(* PLC project drill, Dassault Systèmes ControlBuild 2020 *)
(* stored: creationDateTime 2019-04-23T11:18:46-01:00 *)

CONFIGURATION drill
  VAR_GLOBAL
    generalPanel/powerUpPB AT 7 : BOOL := false;
    generalPanel/startCyclePB AT 8 : BOOL := false;
    generalPanel/emergencyStop AT 9 : BOOL := false;
    generalPanel/batchCycle AT 10 : BOOL := true;
    generalPanel/pieceCycle AT 11 : BOOL := false;
    generalPanel/autoSwitch AT 12 : BOOL := false;
    generalPanel/manualSwitch AT 13 : BOOL := false;
    generalPanel/acknowledgePB AT 15 : BOOL := false;
    generalPanel/powerUpPB/PB AT 7 : BOOL := false;
    generalPanel/powerUpPB/action AT 24 : BOOL := false;
    generalPanel/powerUpPB/timeCounter AT 17 : REAL := 0.0;
    generalPanel/powerUpPB/pulseDuration AT 18 : REAL := 5.0;
    generalPanel/powerUpPB/PBLogic AT 25 : BOOL := true;
    generalPanel/startCyclePB/PB AT 8 : BOOL := false;
    generalPanel/startCyclePB/action AT 26 : BOOL := false;
    generalPanel/startCyclePB/timeCounter AT 19 : REAL := 0.0;
    generalPanel/startCyclePB/pulseDuration AT 20 : REAL := 5.0;
    generalPanel/startCyclePB/PBLogic AT 27 : BOOL := true;
    generalPanel/cycleSwitch/leftVariable AT 11 : BOOL := false;
    generalPanel/cycleSwitch/rightVariable AT 10 : BOOL := true;
    generalPanel/cycleSwitch/leftPosition AT 28 : BOOL := false;
    generalPanel/cycleSwitch/rightPosition AT 29 : BOOL := false;
    generalPanel/modeSwitch/leftVariable AT 12 : BOOL := true;
    generalPanel/modeSwitch/rightVariable AT 13 : BOOL := false;
    generalPanel/modeSwitch/leftPosition AT 30 : BOOL := false;
    generalPanel/modeSwitch/rightPosition AT 31 : BOOL := false;
    generalPanel/acknowledgePB/PB AT 15 : BOOL := false;
    generalPanel/acknowledgePB/action AT 32 : BOOL := false;
    generalPanel/acknowledgePB/timeCounter AT 21 : REAL := 0.0;
    generalPanel/acknowledgePB/pulseDuration AT 22 : REAL := 5.0;
    generalPanel/acknowledgePB/PBLogic AT 33 : BOOL := true;
    generalPanel/emergencyStop/pb AT 9 : BOOL := false;
    generalPanel/emergencyStop/action AT 34 : BOOL := false;
    generalPanel/emergencyStop/PBLogic AT 35 : BOOL := false;
    workingModes/powerUpPB AT 7 : BOOL := false;
    workingModes/startCyclePB AT 8 : BOOL := false;
    workingModes/emergencyStop AT 9 : BOOL := false;
    workingModes/batchCycle AT 10 : BOOL := true;
    workingModes/pieceCycle AT 11 : BOOL := false;
    workingModes/autoSwitch AT 12 : BOOL := false;
    workingModes/manualSwitch AT 13 : BOOL := false;
    workingModes/cycleEnd AT 14 : BOOL := false;
    workingModes/acknowledgePB AT 15 : BOOL := false;
    workingModes/live AT 6 : BOOL := false;
    workingModes/autoMode AT 20 : BOOL := false;
    workingModes/manualMode AT 21 : BOOL := false;
    workingModes/emptyProd AT 17 : BOOL := false;
    workingModes/unitProd AT 18 : BOOL := false;
    workingModes/batchProd AT 19 : BOOL := false;
    workingModes/emergencyState AT 36 : BOOL := false;
    functional/piece AT 16 : BOOL := false;
    functional/emptyProd AT 17 : BOOL := false;
    functional/unitProd AT 18 : BOOL := false;
    functional/batchProd AT 19 : BOOL := false;
    functional/acknowledgePB AT 15 : BOOL := false;
    functional/autoMode AT 20 : BOOL := false;
    functional/manualMode AT 21 : BOOL := false;
    functional/faultyState AT 5 : BOOL := false;
    functional/cycleEnd AT 14 : BOOL := false;
    functional/loadingRequest AT 22 : BOOL := false;
    functional/unloadingRequest AT 23 : BOOL := false;
    functional/functionChart/rotationFault AT 529 : DINT := 0;
    functional/functionChart/downState AT 42 : BOOL := false;
    functional/functionChart/downDeceleration AT 43 : BOOL := false;
    functional/functionChart/topDeceleration AT 44 : BOOL := false;
    functional/functionChart/topState AT 45 : BOOL := false;
    functional/functionChart/motorFault AT 530 : DINT := 0;
    functional/functionChart/clampingFault AT 531 : DINT := 0;
    functional/functionChart/releasingOK AT 46 : BOOL := false;
    functional/functionChart/clampingOK AT 47 : BOOL := false;
    functional/functionChart/emptyProd AT 17 : BOOL := false;
    functional/functionChart/unitProd AT 18 : BOOL := false;
    functional/functionChart/batchProd AT 19 : BOOL := false;
    functional/functionChart/acknowledgePB AT 15 : BOOL := false;
    functional/functionChart/piece AT 16 : BOOL := false;
    functional/functionChart/rotation AT 54 : BOOL := false;
    functional/functionChart/cycleEnd AT 14 : BOOL := false;
    functional/functionChart/movementFault AT 528 : DINT := 0;
    functional/functionChart/loadingRequest AT 22 : BOOL := false;
    functional/functionChart/unloadingRequest AT 23 : BOOL := false;
    functional/functionChart/faultyState AT 5 : BOOL := false;
    functional/functionChart/slowAscent AT 48 : BOOL := false;
    functional/functionChart/fastAscent AT 49 : BOOL := false;
    functional/functionChart/slowDescent AT 50 : BOOL := false;
    functional/functionChart/fastDescent AT 51 : BOOL := false;
    functional/functionChart/releasing AT 52 : BOOL := false;
    functional/functionChart/clamping AT 53 : BOOL := false;
    functional/functionChart/initialCond AT 55 : BOOL := false;
    functional/functionChart/noFaultCond AT 56 : BOOL := false;
    functional/functionChart/cnt AT 532 : DINT := 0;
    functional/functionChart/_X_10 AT 57 : BOOL := true;
    functional/functionChart/_X_11 AT 58 : BOOL := false;
    functional/functionChart/_X_12 AT 59 : BOOL := false;
    functional/functionChart/_X_13 AT 60 : BOOL := false;
    functional/functionChart/_X_14 AT 61 : BOOL := false;
    functional/functionChart/_X_15 AT 62 : BOOL := false;
    functional/functionChart/_X_16 AT 63 : BOOL := false;
    functional/functionChart/_X_17 AT 64 : BOOL := false;
    functional/functionChart/fastDescentDuration AT 533 : DINT := 100;
    functional/functionChart/slowDescentDuration AT 534 : DINT := 50;
    functional/functionChart/fastAscentDuration AT 535 : DINT := 100;
    functional/functionChart/slowAscentDuration AT 536 : DINT := 50;
    functional/descent/slowAscent AT 48 : BOOL := false;
    functional/descent/fastAscent AT 49 : BOOL := false;
    functional/descent/slowDescent AT 50 : BOOL := false;
    functional/descent/fastDescent AT 51 : BOOL := false;
    functional/descent/acknowledgePB AT 15 : BOOL := false;
    functional/descent/autoMode AT 20 : BOOL := false;
    functional/descent/manualMode AT 21 : BOOL := false;
    functional/descent/ascentEnd AT 45 : BOOL := false;
    functional/descent/topDeceleration AT 44 : BOOL := false;
    functional/descent/downDeceleration AT 43 : BOOL := false;
    functional/descent/descentEnd AT 42 : BOOL := false;
    functional/descent/motorFault AT 530 : DINT := 0;
    functional/descent/ascentFunction/acknowledgePB AT 15 : BOOL := false;
    functional/descent/ascentFunction/slowAscent AT 48 : BOOL := false;
    functional/descent/ascentFunction/fastAscent AT 49 : BOOL := false;
    functional/descent/ascentFunction/slowDescent AT 50 : BOOL := false;
    functional/descent/ascentFunction/fastDescent AT 51 : BOOL := false;
    functional/descent/ascentFunction/equipmentFault AT 75 : BOOL := false;
    functional/descent/ascentFunction/motorFault AT 530 : DINT := 0;
    functional/descent/ascentFunction/forward AT 76 : BOOL := false;
    functional/descent/ascentFunction/backward AT 77 : BOOL := false;
    functional/descent/ascentFunction/highSpeed AT 78 : BOOL := false;
    functional/descent/ascentFunction/lowSpeed AT 79 : BOOL := false;
    functional/descent/ascentFunction/_X_10 AT 80 : BOOL := true;
    functional/descent/ascentFunction/_X_11 AT 81 : BOOL := false;
    functional/descent/ascentFunction/_X_20 AT 82 : BOOL := true;
    functional/descent/ascentFunction/_X_21 AT 83 : BOOL := false;
    functional/descent/ascentFunction/_X_30 AT 84 : BOOL := true;
    functional/descent/ascentFunction/_X_31 AT 85 : BOOL := false;
    functional/descent/ascentFunction/_X_40 AT 86 : BOOL := true;
    functional/descent/ascentFunction/_X_41 AT 87 : BOOL := false;
    functional/descent/motorOfTurret/autoMode AT 20 : BOOL := false;
    functional/descent/motorOfTurret/manualMode AT 21 : BOOL := false;
    functional/descent/motorOfTurret/autoFwdCmd AT 76 : BOOL := false;
    functional/descent/motorOfTurret/autoBwdCmd AT 77 : BOOL := false;
    functional/descent/motorOfTurret/autoHSCmd AT 78 : BOOL := false;
    functional/descent/motorOfTurret/autoLSCmd AT 79 : BOOL := false;
    functional/descent/motorOfTurret/acknowledgePB AT 15 : BOOL := false;
    functional/descent/motorOfTurret/speedVal AT 25 : REAL := 0.0;
    functional/descent/motorOfTurret/speedPercent AT 24 : REAL := 0.0;
    functional/descent/motorOfTurret/generalFault AT 75 : BOOL := false;
    functional/descent/motorOfTurret/panel1/forwardPB AT 100 : BOOL := false;
    functional/descent/motorOfTurret/panel1/backwardPB AT 101 : BOOL := false;
    functional/descent/motorOfTurret/panel1/highSpeedPB AT 102 : BOOL := false;
    functional/descent/motorOfTurret/panel1/lowSpeedPB AT 103 : BOOL := false;
    functional/descent/motorOfTurret/panel1/stopPB AT 104 : BOOL := false;
    functional/descent/motorOfTurret/panel1/forwardPB/PB AT 100 : BOOL := false;
    functional/descent/motorOfTurret/panel1/forwardPB/action AT 110 : BOOL := false;
    functional/descent/motorOfTurret/panel1/forwardPB/timeCounter AT 26 : REAL := 0.0;
    functional/descent/motorOfTurret/panel1/forwardPB/pulseDuration AT 27 : REAL := 5.0;
    functional/descent/motorOfTurret/panel1/forwardPB/PBLogic AT 111 : BOOL := true;
    functional/descent/motorOfTurret/panel1/backwardPB/PB AT 101 : BOOL := false;
    functional/descent/motorOfTurret/panel1/backwardPB/action AT 112 : BOOL := false;
    functional/descent/motorOfTurret/panel1/backwardPB/timeCounter AT 28 : REAL := 0.0;
    functional/descent/motorOfTurret/panel1/backwardPB/pulseDuration AT 29 : REAL := 5.0;
    functional/descent/motorOfTurret/panel1/backwardPB/PBLogic AT 113 : BOOL := true;
    functional/descent/motorOfTurret/panel1/speedSwitch/leftVariable AT 102 : BOOL := true;
    functional/descent/motorOfTurret/panel1/speedSwitch/rightVariable AT 103 : BOOL := false;
    functional/descent/motorOfTurret/panel1/speedSwitch/leftPosition AT 114 : BOOL := false;
    functional/descent/motorOfTurret/panel1/speedSwitch/rightPosition AT 115 : BOOL := false;
    functional/descent/motorOfTurret/panel1/stopPB/PB AT 104 : BOOL := false;
    functional/descent/motorOfTurret/panel1/stopPB/action AT 116 : BOOL := false;
    functional/descent/motorOfTurret/panel1/stopPB/timeCounter AT 30 : REAL := 0.0;
    functional/descent/motorOfTurret/panel1/stopPB/pulseDuration AT 31 : REAL := 5.0;
    functional/descent/motorOfTurret/panel1/stopPB/PBLogic AT 117 : BOOL := true;
    functional/descent/motorOfTurret/motor/voltage380 AT 95 : BOOL := true;
    functional/descent/motorOfTurret/motor/cmdSupply AT 94 : BOOL := true;
    functional/descent/motorOfTurret/motor/sensorSupply AT 93 : BOOL := true;
    functional/descent/motorOfTurret/motor/forward AT 96 : BOOL := false;
    functional/descent/motorOfTurret/motor/backward AT 97 : BOOL := false;
    functional/descent/motorOfTurret/motor/highSpeed AT 98 : BOOL := false;
    functional/descent/motorOfTurret/motor/lowSpeed AT 99 : BOOL := false;
    functional/descent/motorOfTurret/motor/forwardFB AT 105 : BOOL := false;
    functional/descent/motorOfTurret/motor/backwardFB AT 106 : BOOL := false;
    functional/descent/motorOfTurret/motor/highSpeedFB AT 107 : BOOL := false;
    functional/descent/motorOfTurret/motor/lowSpeedFB AT 108 : BOOL := false;
    functional/descent/motorOfTurret/motor/thermal AT 109 : BOOL := false;
    functional/descent/motorOfTurret/motor/speedVal AT 25 : REAL := 0.0;
    functional/descent/motorOfTurret/motor/speedPercent AT 24 : REAL := 0.0;
    functional/descent/motorOfTurret/motor/increment AT 32 : REAL := 0.0;
    functional/descent/motorOfTurret/motor/memoFwd AT 118 : BOOL := false;
    functional/descent/motorOfTurret/motor/memoBwd AT 119 : BOOL := false;
    functional/descent/motorOfTurret/motor/memoHighSpeed AT 120 : BOOL := false;
    functional/descent/motorOfTurret/motor/memoLowSpeed AT 121 : BOOL := false;
    functional/descent/motorOfTurret/motor/FwdHsState AT 122 : BOOL := false;
    functional/descent/motorOfTurret/motor/FwdLsState AT 123 : BOOL := false;
    functional/descent/motorOfTurret/motor/BwdHsState AT 124 : BOOL := false;
    functional/descent/motorOfTurret/motor/BwdLsState AT 125 : BOOL := false;
    functional/descent/motorOfTurret/motor/wantedSpeed AT 33 : REAL := 0.0;
    functional/descent/motorOfTurret/motor/nominalTime AT 34 : REAL := 0.05;
    functional/descent/motorOfTurret/motor/thermalLogic AT 126 : BOOL := false;
    functional/descent/motorOfTurret/motor/fwdFbLogic AT 127 : BOOL := true;
    functional/descent/motorOfTurret/motor/bwdFbLogic AT 128 : BOOL := true;
    functional/descent/motorOfTurret/motor/highSpeedFbLogic AT 129 : BOOL := true;
    functional/descent/motorOfTurret/motor/lowSpeedFbLogic AT 130 : BOOL := true;
    functional/descent/motorOfTurret/motor/nominalLowSpeed AT 35 : REAL := 100.0;
    functional/descent/motorOfTurret/motor/nominalHighSpeed AT 36 : REAL := 200.0;
    functional/descent/motorOfTurret/motor/d_locking AT 131 : BOOL := false;
    functional/descent/motorOfTurret/motor/v_d_locking AT 37 : REAL := 0.5;
    functional/descent/motorOfTurret/motor/d_electrical AT 132 : BOOL := false;
    functional/descent/motorOfTurret/motor/v_d_electrical AT 133 : BOOL := false;
    functional/descent/motorOfTurret/motor/d_forwardFB AT 134 : BOOL := false;
    functional/descent/motorOfTurret/motor/v_d_forwardFB AT 135 : BOOL := false;
    functional/descent/motorOfTurret/motor/d_highSpeedFB AT 136 : BOOL := false;
    functional/descent/motorOfTurret/motor/v_d_highSpeedFB AT 137 : BOOL := false;
    functional/descent/motorOfTurret/motor/d_lowSpeedFB AT 138 : BOOL := false;
    functional/descent/motorOfTurret/motor/v_d_lowSpeedFB AT 139 : BOOL := false;
    functional/descent/motorOfTurret/motor/d_backwardFB AT 140 : BOOL := false;
    functional/descent/motorOfTurret/motor/v_d_backwardFB AT 141 : BOOL := false;
    functional/descent/motorOfTurret/cmdOfMotor/autoMode AT 20 : BOOL := false;
    functional/descent/motorOfTurret/cmdOfMotor/manualMode AT 21 : BOOL := false;
    functional/descent/motorOfTurret/cmdOfMotor/autoFwdCmd AT 76 : BOOL := false;
    functional/descent/motorOfTurret/cmdOfMotor/autoBwdCmd AT 77 : BOOL := false;
    functional/descent/motorOfTurret/cmdOfMotor/autoHSCmd AT 78 : BOOL := false;
    functional/descent/motorOfTurret/cmdOfMotor/autoLSCmd AT 79 : BOOL := false;
    functional/descent/motorOfTurret/cmdOfMotor/forwardPB AT 100 : BOOL := false;
    functional/descent/motorOfTurret/cmdOfMotor/backwardPB AT 101 : BOOL := false;
    functional/descent/motorOfTurret/cmdOfMotor/highSpeedPB AT 102 : BOOL := false;
    functional/descent/motorOfTurret/cmdOfMotor/lowSpeedPB AT 103 : BOOL := false;
    functional/descent/motorOfTurret/cmdOfMotor/stopPB AT 104 : BOOL := false;
    functional/descent/motorOfTurret/cmdOfMotor/forwardFB AT 105 : BOOL := false;
    functional/descent/motorOfTurret/cmdOfMotor/backwardFB AT 106 : BOOL := false;
    functional/descent/motorOfTurret/cmdOfMotor/highSpeedFB AT 107 : BOOL := false;
    functional/descent/motorOfTurret/cmdOfMotor/lowSpeedFB AT 108 : BOOL := false;
    functional/descent/motorOfTurret/cmdOfMotor/thermalFB AT 109 : BOOL := false;
    functional/descent/motorOfTurret/cmdOfMotor/acknowledgePB AT 15 : BOOL := false;
    functional/descent/motorOfTurret/cmdOfMotor/forwardCmd AT 96 : BOOL := false;
    functional/descent/motorOfTurret/cmdOfMotor/backwardCmd AT 97 : BOOL := false;
    functional/descent/motorOfTurret/cmdOfMotor/highSpeedCmd AT 98 : BOOL := false;
    functional/descent/motorOfTurret/cmdOfMotor/lowSpeedCmd AT 99 : BOOL := false;
    functional/descent/motorOfTurret/cmdOfMotor/generalFault AT 75 : BOOL := false;
    functional/descent/motorOfTurret/cmdOfMotor/actions/autoMode AT 20 : BOOL := false;
    functional/descent/motorOfTurret/cmdOfMotor/actions/manualMode AT 21 : BOOL := false;
    functional/descent/motorOfTurret/cmdOfMotor/actions/autoFwdCmd AT 76 : BOOL := false;
    functional/descent/motorOfTurret/cmdOfMotor/actions/autoBwdCmd AT 77 : BOOL := false;
    functional/descent/motorOfTurret/cmdOfMotor/actions/autoHSCmd AT 78 : BOOL := false;
    functional/descent/motorOfTurret/cmdOfMotor/actions/autoLSCmd AT 79 : BOOL := false;
    functional/descent/motorOfTurret/cmdOfMotor/actions/forwardPB AT 100 : BOOL := false;
    functional/descent/motorOfTurret/cmdOfMotor/actions/backwardPB AT 101 : BOOL := false;
    functional/descent/motorOfTurret/cmdOfMotor/actions/highSpeedPB AT 102 : BOOL := false;
    functional/descent/motorOfTurret/cmdOfMotor/actions/lowSpeedPB AT 103 : BOOL := false;
    functional/descent/motorOfTurret/cmdOfMotor/actions/stopPB AT 104 : BOOL := false;
    functional/descent/motorOfTurret/cmdOfMotor/actions/generalFault AT 75 : BOOL := false;
    functional/descent/motorOfTurret/cmdOfMotor/actions/forwardCmd AT 96 : BOOL := false;
    functional/descent/motorOfTurret/cmdOfMotor/actions/backwardCmd AT 97 : BOOL := false;
    functional/descent/motorOfTurret/cmdOfMotor/actions/highSpeedCmd AT 98 : BOOL := false;
    functional/descent/motorOfTurret/cmdOfMotor/actions/lowSpeedCmd AT 99 : BOOL := false;
    functional/descent/motorOfTurret/cmdOfMotor/faults1/forwardCmd AT 96 : BOOL := false;
    functional/descent/motorOfTurret/cmdOfMotor/faults1/backwardCmd AT 97 : BOOL := false;
    functional/descent/motorOfTurret/cmdOfMotor/faults1/highSpeedCmd AT 98 : BOOL := false;
    functional/descent/motorOfTurret/cmdOfMotor/faults1/lowSpeedCmd AT 99 : BOOL := false;
    functional/descent/motorOfTurret/cmdOfMotor/faults1/thermalFB AT 109 : BOOL := false;
    functional/descent/motorOfTurret/cmdOfMotor/faults1/forwardFB AT 105 : BOOL := false;
    functional/descent/motorOfTurret/cmdOfMotor/faults1/backwardFB AT 106 : BOOL := false;
    functional/descent/motorOfTurret/cmdOfMotor/faults1/highSpeedFB AT 107 : BOOL := false;
    functional/descent/motorOfTurret/cmdOfMotor/faults1/lowSpeedFB AT 108 : BOOL := false;
    functional/descent/motorOfTurret/cmdOfMotor/faults1/acknowledgePB AT 15 : BOOL := false;
    functional/descent/motorOfTurret/cmdOfMotor/faults1/generalFault AT 75 : BOOL := false;
    functional/descent/motorOfTurret/cmdOfMotor/faults1/thermalFault AT 142 : BOOL := false;
    functional/descent/motorOfTurret/cmdOfMotor/faults1/forwardFBFault AT 143 : BOOL := false;
    functional/descent/motorOfTurret/cmdOfMotor/faults1/backwardFBFault AT 144 : BOOL := false;
    functional/descent/turret/speed AT 25 : REAL := 0.0;
    functional/descent/turret/forward AT 76 : BOOL := false;
    functional/descent/turret/backward AT 77 : BOOL := false;
    functional/descent/turret/highSpeed AT 78 : BOOL := false;
    functional/descent/turret/lowSpeed AT 79 : BOOL := false;
    functional/descent/turret/axlePosition AT 23 : REAL := 0.0;
    functional/descent/turret/forwardEnd AT 42 : BOOL := false;
    functional/descent/turret/forwardDeceleration AT 43 : BOOL := false;
    functional/descent/turret/backwardDeceleration AT 44 : BOOL := false;
    functional/descent/turret/backwardEnd AT 45 : BOOL := false;
    functional/descent/turret/speedIncrement AT 38 : REAL := 0.0;
    functional/descent/turret/lockingFault AT 149 : BOOL := false;
    functional/descent/turret/forwardEndFault AT 150 : BOOL := false;
    functional/descent/turret/forwardEndValue AT 151 : BOOL := false;
    functional/descent/turret/forwardDecelerationFault AT 152 : BOOL := false;
    functional/descent/turret/forwardDecelerationValue AT 153 : BOOL := false;
    functional/descent/turret/backwardDecelerationFault AT 154 : BOOL := false;
    functional/descent/turret/backwardDecelerationValue AT 155 : BOOL := false;
    functional/descent/turret/backwardEndFault AT 156 : BOOL := false;
    functional/descent/turret/backwardEndValue AT 157 : BOOL := false;
    functional/descent/turret/axleLength AT 39 : REAL := 100.0;
    functional/descent/turret/forwardDecelerationPosition AT 556 : DINT := 70;
    functional/descent/turret/backwardDecelerationPosition AT 557 : DINT := 30;
    functional/descent/turret/range AT 558 : DINT := 10;
    functional/clamping/acknowledgePB AT 15 : BOOL := false;
    functional/clamping/autoMode AT 20 : BOOL := false;
    functional/clamping/manualMode AT 21 : BOOL := false;
    functional/clamping/releasing AT 52 : BOOL := false;
    functional/clamping/clamping AT 53 : BOOL := false;
    functional/clamping/clampingOK AT 47 : BOOL := false;
    functional/clamping/releasingOK AT 46 : BOOL := false;
    functional/clamping/clampingFault AT 531 : DINT := 0;
    functional/clamping/clampingFunction/acknowledgePB AT 15 : BOOL := false;
    functional/clamping/clampingFunction/releasing AT 52 : BOOL := false;
    functional/clamping/clampingFunction/clamping AT 53 : BOOL := false;
    functional/clamping/clampingFunction/rightUnlocked AT 158 : BOOL := false;
    functional/clamping/clampingFunction/rightLocked AT 159 : BOOL := false;
    functional/clamping/clampingFunction/leftUnlocked AT 160 : BOOL := false;
    functional/clamping/clampingFunction/leftLocked AT 161 : BOOL := false;
    functional/clamping/clampingFunction/rightFault AT 162 : BOOL := false;
    functional/clamping/clampingFunction/leftFault AT 163 : BOOL := false;
    functional/clamping/clampingFunction/clampingOK AT 47 : BOOL := false;
    functional/clamping/clampingFunction/releasingOK AT 46 : BOOL := false;
    functional/clamping/clampingFunction/clampingFault AT 531 : DINT := 0;
    functional/clamping/clampingFunction/rightLocking AT 165 : BOOL := false;
    functional/clamping/clampingFunction/leftLocking AT 164 : BOOL := false;
    functional/clamping/clampingFunction/_X_10 AT 166 : BOOL := true;
    functional/clamping/clampingFunction/_X_11 AT 167 : BOOL := false;
    functional/clamping/clampingFunction/_X_12 AT 168 : BOOL := false;
    functional/clamping/clampingFunction/_X_13 AT 169 : BOOL := false;
    functional/clamping/clampingFunction/_X_14 AT 170 : BOOL := false;
    functional/clamping/clampingFunction/clampingDuration AT 559 : DINT := 110;
    functional/clamping/clampingFunction/releasingDuration AT 560 : DINT := 110;
    functional/clamping/leftJack/acknowledgePB AT 15 : BOOL := false;
    functional/clamping/leftJack/autoMode AT 20 : BOOL := false;
    functional/clamping/leftJack/manualMode AT 21 : BOOL := false;
    functional/clamping/leftJack/autoWorkCmd AT 164 : BOOL := false;
    functional/clamping/leftJack/generalFault AT 163 : BOOL := false;
    functional/clamping/leftJack/inletSensor AT 160 : BOOL := false;
    functional/clamping/leftJack/outletSensor AT 161 : BOOL := false;
    functional/clamping/leftJack/rodPosition AT 45 : REAL := 0.0;
    functional/clamping/leftJack/rodPercent AT 44 : REAL := 0.0;
    functional/clamping/leftJack/incrementValue AT 43 : REAL := 0.0;
    functional/clamping/leftJack/panel1/valveWorkPB AT 177 : BOOL := false;
    functional/clamping/leftJack/panel1/switch/variable AT 177 : BOOL := false;
    functional/clamping/leftJack/panel1/switch/leftPosition AT 179 : BOOL := false;
    functional/clamping/leftJack/panel1/switch/rightPosition AT 180 : BOOL := false;
    functional/clamping/leftJack/cmdOfJack/autoMode AT 20 : BOOL := false;
    functional/clamping/leftJack/cmdOfJack/manualMode AT 21 : BOOL := false;
    functional/clamping/leftJack/cmdOfJack/autoWorkCmd AT 164 : BOOL := false;
    functional/clamping/leftJack/cmdOfJack/valveWorkPB AT 177 : BOOL := false;
    functional/clamping/leftJack/cmdOfJack/outletSensor AT 161 : BOOL := false;
    functional/clamping/leftJack/cmdOfJack/inletSensor AT 160 : BOOL := false;
    functional/clamping/leftJack/cmdOfJack/acknowledgePB AT 15 : BOOL := false;
    functional/clamping/leftJack/cmdOfJack/workCmd AT 178 : BOOL := false;
    functional/clamping/leftJack/cmdOfJack/generalFault AT 163 : BOOL := false;
    functional/clamping/leftJack/cmdOfJack/actions/autoMode AT 20 : BOOL := false;
    functional/clamping/leftJack/cmdOfJack/actions/manualMode AT 21 : BOOL := false;
    functional/clamping/leftJack/cmdOfJack/actions/autoWorkCmd AT 164 : BOOL := false;
    functional/clamping/leftJack/cmdOfJack/actions/valveWorkPB AT 177 : BOOL := false;
    functional/clamping/leftJack/cmdOfJack/actions/generalFault AT 163 : BOOL := false;
    functional/clamping/leftJack/cmdOfJack/actions/workCmd AT 178 : BOOL := false;
    functional/clamping/leftJack/cmdOfJack/faults1/workCmd AT 178 : BOOL := false;
    functional/clamping/leftJack/cmdOfJack/faults1/outletSensor AT 161 : BOOL := false;
    functional/clamping/leftJack/cmdOfJack/faults1/inletSensor AT 160 : BOOL := false;
    functional/clamping/leftJack/cmdOfJack/faults1/acknowledgePB AT 15 : BOOL := false;
    functional/clamping/leftJack/cmdOfJack/faults1/generalFault AT 163 : BOOL := false;
    functional/clamping/leftJack/cmdOfJack/faults1/discordanceFault AT 181 : BOOL := false;
    functional/clamping/leftJack/cmdOfJack/faults1/outletSensorFault AT 182 : BOOL := false;
    functional/clamping/leftJack/cmdOfJack/faults1/inletSensorFault AT 183 : BOOL := false;
    functional/clamping/leftJack/cmdOfJack/faults1/presetMvt AT 562 : TIME := T#0h0m10s0ms;
    functional/clamping/leftJack/cmdOfJack/faults1/presetDiscordance AT 566 : TIME := T#0h0m0s200ms;
    functional/clamping/leftJack/jack/energy AT 176 : BOOL := true;
    functional/clamping/leftJack/jack/cmdSupply AT 175 : BOOL := true;
    functional/clamping/leftJack/jack/sensorSupply AT 174 : BOOL := true;
    functional/clamping/leftJack/jack/valveWork AT 178 : BOOL := false;
    functional/clamping/leftJack/jack/outletSensor AT 161 : BOOL := false;
    functional/clamping/leftJack/jack/inletSensor AT 160 : BOOL := false;
    functional/clamping/leftJack/jack/rodPosition AT 45 : REAL := 0.0;
    functional/clamping/leftJack/jack/rodPercent AT 44 : REAL := 0.0;
    functional/clamping/leftJack/jack/incrementValue AT 43 : REAL := 0.0;
    functional/clamping/leftJack/jack/slidePosition AT 594 : DINT := 0;
    functional/clamping/leftJack/jack/pipeWork AT 190 : BOOL := false;
    functional/clamping/leftJack/jack/pipeRest AT 191 : BOOL := false;
    functional/clamping/leftJack/jack/increment AT 46 : REAL := 0.0;
    functional/clamping/leftJack/jack/outletSensorLogic AT 192 : BOOL := true;
    functional/clamping/leftJack/jack/inletSensorLogic AT 193 : BOOL := true;
    functional/clamping/leftJack/jack/rodLength AT 47 : REAL := 1000.0;
    functional/clamping/leftJack/jack/time2extend AT 48 : REAL := 1.0;
    functional/clamping/leftJack/jack/d_locking AT 194 : BOOL := false;
    functional/clamping/leftJack/jack/v_d_locking AT 49 : REAL := 2.0;
    functional/clamping/leftJack/jack/d_inletSensor AT 195 : BOOL := false;
    functional/clamping/leftJack/jack/v_d_inletSensor AT 196 : BOOL := false;
    functional/clamping/leftJack/jack/d_outletSensor AT 197 : BOOL := false;
    functional/clamping/leftJack/jack/v_d_outletSensor AT 198 : BOOL := false;
    functional/clamping/rightJack/acknowledgePB AT 15 : BOOL := false;
    functional/clamping/rightJack/autoMode AT 20 : BOOL := false;
    functional/clamping/rightJack/manualMode AT 21 : BOOL := false;
    functional/clamping/rightJack/autoWorkCmd AT 165 : BOOL := false;
    functional/clamping/rightJack/generalFault AT 162 : BOOL := false;
    functional/clamping/rightJack/inletSensor AT 158 : BOOL := false;
    functional/clamping/rightJack/outletSensor AT 159 : BOOL := false;
    functional/clamping/rightJack/rodPosition AT 42 : REAL := 0.0;
    functional/clamping/rightJack/rodPercent AT 41 : REAL := 0.0;
    functional/clamping/rightJack/incrementValue AT 40 : REAL := 0.0;
    functional/clamping/rightJack/panel1/valveWorkPB AT 202 : BOOL := false;
    functional/clamping/rightJack/panel1/switch/variable AT 202 : BOOL := false;
    functional/clamping/rightJack/panel1/switch/leftPosition AT 204 : BOOL := false;
    functional/clamping/rightJack/panel1/switch/rightPosition AT 205 : BOOL := false;
    functional/clamping/rightJack/cmdOfJack/autoMode AT 20 : BOOL := false;
    functional/clamping/rightJack/cmdOfJack/manualMode AT 21 : BOOL := false;
    functional/clamping/rightJack/cmdOfJack/autoWorkCmd AT 165 : BOOL := false;
    functional/clamping/rightJack/cmdOfJack/valveWorkPB AT 202 : BOOL := false;
    functional/clamping/rightJack/cmdOfJack/outletSensor AT 159 : BOOL := false;
    functional/clamping/rightJack/cmdOfJack/inletSensor AT 158 : BOOL := false;
    functional/clamping/rightJack/cmdOfJack/acknowledgePB AT 15 : BOOL := false;
    functional/clamping/rightJack/cmdOfJack/workCmd AT 203 : BOOL := false;
    functional/clamping/rightJack/cmdOfJack/generalFault AT 162 : BOOL := false;
    functional/clamping/rightJack/cmdOfJack/actions/autoMode AT 20 : BOOL := false;
    functional/clamping/rightJack/cmdOfJack/actions/manualMode AT 21 : BOOL := false;
    functional/clamping/rightJack/cmdOfJack/actions/autoWorkCmd AT 165 : BOOL := false;
    functional/clamping/rightJack/cmdOfJack/actions/valveWorkPB AT 202 : BOOL := false;
    functional/clamping/rightJack/cmdOfJack/actions/generalFault AT 162 : BOOL := false;
    functional/clamping/rightJack/cmdOfJack/actions/workCmd AT 203 : BOOL := false;
    functional/clamping/rightJack/cmdOfJack/faults1/workCmd AT 203 : BOOL := false;
    functional/clamping/rightJack/cmdOfJack/faults1/outletSensor AT 159 : BOOL := false;
    functional/clamping/rightJack/cmdOfJack/faults1/inletSensor AT 158 : BOOL := false;
    functional/clamping/rightJack/cmdOfJack/faults1/acknowledgePB AT 15 : BOOL := false;
    functional/clamping/rightJack/cmdOfJack/faults1/generalFault AT 162 : BOOL := false;
    functional/clamping/rightJack/cmdOfJack/faults1/discordanceFault AT 206 : BOOL := false;
    functional/clamping/rightJack/cmdOfJack/faults1/outletSensorFault AT 207 : BOOL := false;
    functional/clamping/rightJack/cmdOfJack/faults1/inletSensorFault AT 208 : BOOL := false;
    functional/clamping/rightJack/cmdOfJack/faults1/presetMvt AT 595 : TIME := T#0h0m10s0ms;
    functional/clamping/rightJack/cmdOfJack/faults1/presetDiscordance AT 599 : TIME := T#0h0m0s200ms;
    functional/clamping/rightJack/jack/energy AT 201 : BOOL := true;
    functional/clamping/rightJack/jack/cmdSupply AT 200 : BOOL := true;
    functional/clamping/rightJack/jack/sensorSupply AT 199 : BOOL := true;
    functional/clamping/rightJack/jack/valveWork AT 203 : BOOL := false;
    functional/clamping/rightJack/jack/outletSensor AT 159 : BOOL := false;
    functional/clamping/rightJack/jack/inletSensor AT 158 : BOOL := false;
    functional/clamping/rightJack/jack/rodPosition AT 42 : REAL := 0.0;
    functional/clamping/rightJack/jack/rodPercent AT 41 : REAL := 0.0;
    functional/clamping/rightJack/jack/incrementValue AT 40 : REAL := 0.0;
    functional/clamping/rightJack/jack/slidePosition AT 627 : DINT := 0;
    functional/clamping/rightJack/jack/pipeWork AT 215 : BOOL := false;
    functional/clamping/rightJack/jack/pipeRest AT 216 : BOOL := false;
    functional/clamping/rightJack/jack/increment AT 50 : REAL := 0.0;
    functional/clamping/rightJack/jack/outletSensorLogic AT 217 : BOOL := true;
    functional/clamping/rightJack/jack/inletSensorLogic AT 218 : BOOL := true;
    functional/clamping/rightJack/jack/rodLength AT 51 : REAL := 1000.0;
    functional/clamping/rightJack/jack/time2extend AT 52 : REAL := 1.0;
    functional/clamping/rightJack/jack/d_locking AT 219 : BOOL := false;
    functional/clamping/rightJack/jack/v_d_locking AT 53 : REAL := 2.0;
    functional/clamping/rightJack/jack/d_inletSensor AT 220 : BOOL := false;
    functional/clamping/rightJack/jack/v_d_inletSensor AT 221 : BOOL := false;
    functional/clamping/rightJack/jack/d_outletSensor AT 222 : BOOL := false;
    functional/clamping/rightJack/jack/v_d_outletSensor AT 223 : BOOL := false;
    functional/spindle/rotationFunction AT 54 : BOOL := false;
    functional/spindle/acknowledgePB AT 15 : BOOL := false;
    functional/spindle/autoMode AT 20 : BOOL := false;
    functional/spindle/manualMode AT 21 : BOOL := false;
    functional/spindle/rotationFault AT 529 : DINT := 0;
    functional/spindle/spindle/rotation AT 54 : BOOL := false;
    functional/spindle/spindle/acknowledgePB AT 15 : BOOL := false;
    functional/spindle/spindle/equipmentFault AT 224 : BOOL := false;
    functional/spindle/spindle/contactor AT 225 : BOOL := false;
    functional/spindle/spindle/rotationFault AT 529 : DINT := 0;
    functional/spindle/spindle/_X_10 AT 226 : BOOL := true;
    functional/spindle/spindle/_X_11 AT 227 : BOOL := false;
    functional/spindle/spindleMotor/autoMode AT 20 : BOOL := false;
    functional/spindle/spindleMotor/manualMode AT 21 : BOOL := false;
    functional/spindle/spindleMotor/autoCmd AT 225 : BOOL := false;
    functional/spindle/spindleMotor/acknowledgePB AT 15 : BOOL := false;
    functional/spindle/spindleMotor/speedVal AT 55 : REAL := 0.0;
    functional/spindle/spindleMotor/speedPercent AT 54 : REAL := 0.0;
    functional/spindle/spindleMotor/generalFault AT 224 : BOOL := false;
    functional/spindle/spindleMotor/panel1/forwardPB AT 236 : BOOL := false;
    functional/spindle/spindleMotor/panel1/stopPB AT 237 : BOOL := false;
    functional/spindle/spindleMotor/panel1/forwardPB/PB AT 236 : BOOL := false;
    functional/spindle/spindleMotor/panel1/forwardPB/action AT 238 : BOOL := false;
    functional/spindle/spindleMotor/panel1/forwardPB/timeCounter AT 56 : REAL := 0.0;
    functional/spindle/spindleMotor/panel1/forwardPB/pulseDuration AT 57 : REAL := 5.0;
    functional/spindle/spindleMotor/panel1/forwardPB/PBLogic AT 239 : BOOL := true;
    functional/spindle/spindleMotor/panel1/stopPB/PB AT 237 : BOOL := false;
    functional/spindle/spindleMotor/panel1/stopPB/action AT 240 : BOOL := false;
    functional/spindle/spindleMotor/panel1/stopPB/timeCounter AT 58 : REAL := 0.0;
    functional/spindle/spindleMotor/panel1/stopPB/pulseDuration AT 59 : REAL := 5.0;
    functional/spindle/spindleMotor/panel1/stopPB/PBLogic AT 241 : BOOL := true;
    functional/spindle/spindleMotor/motor/voltage380 AT 232 : BOOL := true;
    functional/spindle/spindleMotor/motor/cmdSupply AT 231 : BOOL := true;
    functional/spindle/spindleMotor/motor/sensorSupply AT 230 : BOOL := true;
    functional/spindle/spindleMotor/motor/forward AT 233 : BOOL := false;
    functional/spindle/spindleMotor/motor/forwardFB AT 234 : BOOL := false;
    functional/spindle/spindleMotor/motor/thermal AT 235 : BOOL := false;
    functional/spindle/spindleMotor/motor/speedVal AT 55 : REAL := 0.0;
    functional/spindle/spindleMotor/motor/speedPercent AT 54 : REAL := 0.0;
    functional/spindle/spindleMotor/motor/increment AT 60 : REAL := 0.0;
    functional/spindle/spindleMotor/motor/memoFwd AT 242 : BOOL := false;
    functional/spindle/spindleMotor/motor/forwardState AT 243 : BOOL := false;
    functional/spindle/spindleMotor/motor/wantedSpeed AT 61 : REAL := 0.0;
    functional/spindle/spindleMotor/motor/nominalSpeed AT 62 : REAL := 5000.0;
    functional/spindle/spindleMotor/motor/nominalTime AT 63 : REAL := 0.5;
    functional/spindle/spindleMotor/motor/thermalLogic AT 244 : BOOL := false;
    functional/spindle/spindleMotor/motor/feedbackLogic AT 245 : BOOL := true;
    functional/spindle/spindleMotor/motor/d_locking AT 246 : BOOL := false;
    functional/spindle/spindleMotor/motor/v_d_locking AT 64 : REAL := 0.0;
    functional/spindle/spindleMotor/motor/d_feedback AT 247 : BOOL := false;
    functional/spindle/spindleMotor/motor/v_d_feedback AT 248 : BOOL := false;
    functional/spindle/spindleMotor/motor/d_electrical AT 249 : BOOL := false;
    functional/spindle/spindleMotor/motor/v_d_electrical AT 250 : BOOL := false;
    functional/spindle/spindleMotor/cmdOfMotor/autoMode AT 20 : BOOL := false;
    functional/spindle/spindleMotor/cmdOfMotor/manualMode AT 21 : BOOL := false;
    functional/spindle/spindleMotor/cmdOfMotor/autoCmd AT 225 : BOOL := false;
    functional/spindle/spindleMotor/cmdOfMotor/forwardFB AT 234 : BOOL := false;
    functional/spindle/spindleMotor/cmdOfMotor/thermalFB AT 235 : BOOL := false;
    functional/spindle/spindleMotor/cmdOfMotor/forwardPB AT 236 : BOOL := false;
    functional/spindle/spindleMotor/cmdOfMotor/stopPB AT 237 : BOOL := false;
    functional/spindle/spindleMotor/cmdOfMotor/acknowledgePB AT 15 : BOOL := false;
    functional/spindle/spindleMotor/cmdOfMotor/forwardCmd AT 233 : BOOL := false;
    functional/spindle/spindleMotor/cmdOfMotor/generalFault AT 224 : BOOL := false;
    functional/spindle/spindleMotor/cmdOfMotor/actions/autoMode AT 20 : BOOL := false;
    functional/spindle/spindleMotor/cmdOfMotor/actions/manualMode AT 21 : BOOL := false;
    functional/spindle/spindleMotor/cmdOfMotor/actions/autoCmd AT 225 : BOOL := false;
    functional/spindle/spindleMotor/cmdOfMotor/actions/forwardPB AT 236 : BOOL := false;
    functional/spindle/spindleMotor/cmdOfMotor/actions/stopPB AT 237 : BOOL := false;
    functional/spindle/spindleMotor/cmdOfMotor/actions/generalFault AT 224 : BOOL := false;
    functional/spindle/spindleMotor/cmdOfMotor/actions/forwardCmd AT 233 : BOOL := false;
    functional/spindle/spindleMotor/cmdOfMotor/faults1/forwardCmd AT 233 : BOOL := false;
    functional/spindle/spindleMotor/cmdOfMotor/faults1/thermalFB AT 235 : BOOL := false;
    functional/spindle/spindleMotor/cmdOfMotor/faults1/forwardFB AT 234 : BOOL := false;
    functional/spindle/spindleMotor/cmdOfMotor/faults1/acknowledgePB AT 15 : BOOL := false;
    functional/spindle/spindleMotor/cmdOfMotor/faults1/generalFault AT 224 : BOOL := false;
    functional/spindle/spindleMotor/cmdOfMotor/faults1/thermalFault AT 251 : BOOL := false;
    functional/spindle/spindleMotor/cmdOfMotor/faults1/forwardFault AT 252 : BOOL := false;
    load/loadingRequest AT 22 : BOOL := false;
    load/unloadingRequest AT 23 : BOOL := false;
    load/piece AT 16 : BOOL := false;
    load/count AT 637 : DINT := 0;
    load/loadingDuration AT 638 : DINT := 10;
  END_VAR
END_CONFIGURATION
